{attribute 'qualified_only'}
{attribute 'strict'}
{attribute 'to_string'}
TYPE E_SawtoothType  :
(
    Rising := 0,    // Rising sawtooth (ramp up)
    Falling := 1    // Falling sawtooth (ramp down)
);
END_TYPE

(* stored: Version 1.1.0.1
   DUT E_SawtoothType: Id {5811fdc9-7122-4647-b081-247cb36b0893} *)
